Fanuc KAREL source: kt00010.KL

-- PROVISIONAL review KL for V940-1; original PC SHA256 4f19c5a5a5380058b5d0cad27bec187c8a03611e7a19c52fa69866a299b993dd
-- Incomplete behavior may be omitted. Consult companion uncertainty JSON. Do not deploy.
PROGRAM KT00010
%NOLOCKGROUP
VAR
  R1 : REAL
  I2 : INTEGER
  OUT : REAL
BEGIN
  -- V9_ZERO_TABLE_METADATA_HINT layout=0001; no indexed target words; source/name/runtime held
  -- UNRESOLVED_PC offsets 5-16; opcodes 2E,23
  -- UNRESOLVED_PC offsets 21-32; opcodes 2E,23
  -- UNRESOLVED_PC offsets 37-57; opcodes 21,21,64,69,23
  -- UNRESOLVED_PC offsets 62-66; opcodes 7F
END KT00010
